{library PUBLIC}
TYPE ABB_SYNC_FUNCTION_NUMBER :(
(* Set variable values
	ParameterW is the new value *)
	ABB_SYNC_FUNCTION_SET_X:=11,
	ABB_SYNC_FUNCTION_SET_Y:=12,
	ABB_SYNC_FUNCTION_SET_Z:=13,
	ABB_SYNC_FUNCTION_SET_RX:=14,
	ABB_SYNC_FUNCTION_SET_RY:=15,
	ABB_SYNC_FUNCTION_SET_RZ:=16,

(* Get variable values *)
	ABB_SYNC_FUNCTION_GET_X:=21,
	ABB_SYNC_FUNCTION_GET_Y:=22,
	ABB_SYNC_FUNCTION_GET_Z:=23,
	ABB_SYNC_FUNCTION_GET_RX:=24,
	ABB_SYNC_FUNCTION_GET_RY:=25,
	ABB_SYNC_FUNCTION_GET_RZ:=26,

(* Set pneumatic valve value
	ParameterB=1 or 0 *)
	ABB_SYNC_SET_VALVE1:=31,
	ABB_SYNC_SET_VALVE2:=32,
	ABB_SYNC_SET_VALVE3:=33,

	ABB_SYNC_GET_VALVE1:=41,
	ABB_SYNC_GET_VALVE2:=42,
	ABB_SYNC_GET_VALVE3:=43,

	ABB_SYNC_READ_DI:=101,
	ABB_SYNC_WRITE_DO:=102

);
END_TYPE

(* stored: Version 1.1.0.1, ProductVersion 3.1.4024.2
   EnumerationTextList ABB_SYNC_FUNCTION_NUMBER: Id {93d3a9a4-6e1c-4320-a550-3e49b577f2a9} *)
